PROGRAM MAIN
VAR
	fValue : LREAL;
	nValue : UDINT;
END_VAR

END_PROGRAM

(* stored: Version 1.1.0.1, ProductVersion 3.1.4024.9
   POU MAIN: Id {36ee831a-606f-4333-b640-1a57f50c75a5}, SpecialFunc None *)
